FUNCTION_BLOCK FB_SoftWash IMPLEMENTS I_WashStrategy
VAR
	 stSettings : ST_WashSettings; 
    bStarted : BOOL := FALSE; 
END_VAR

METHOD FB_init : BOOL
VAR_INPUT
	bInitRetains : BOOL; // if TRUE, the retain variables are initialized (warm start / cold start)
	bInCopyCode : BOOL;  // if TRUE, the instance afterwards gets moved into the copy code (online change)
END_VAR
IF stSettings.sDescription = '' THEN 
    stSettings.rTemperature  := GVL_WashConstants.SOFT_TEMP; 
    stSettings.nSpinSpeed    := GVL_WashConstants.SOFT_SPIN; 
    stSettings.tWashDuration := GVL_WashConstants.SOFT_WASH_TIME; 
    stSettings.sDescription  := GVL_WashConstants.SOFT_DESC; 

END_IF 

 FB_init := TRUE;
END_METHOD

{warning 'add method implementation '}
METHOD GetDuration : TIME
  GetDuration := stSettings.tWashDuration;
END_METHOD

{warning 'add method implementation '}
METHOD GetProgramName : STRING
 GetProgramName := 'SOFT';
END_METHOD

{warning 'add method implementation '}
METHOD GetSettings : ST_WashSettings
  GetSettings := stSettings;
END_METHOD

{warning 'add method implementation '}
METHOD Start : BOOL
bStarted := TRUE; 
Start     := TRUE;
END_METHOD

END_FUNCTION_BLOCK

(* stored: Version 1.1.0.1, ProductVersion 3.1.4024.16
   POU FB_SoftWash: Id {20098e3f-b3d7-4b4d-bf5b-8d6ee14faa53}, SpecialFunc None
   Method FB_init: Id {a4b3b9de-443f-4248-aed5-d62c01d2d711}
   Method GetDuration: Id {87afdd7e-b00b-4cfb-a9ab-b46c0c02e1ff}
   Method GetProgramName: Id {55729a0a-7107-4950-a342-812a8f56501f}
   Method GetSettings: Id {81cfdbe6-36fa-42dd-a16c-4f0e926ac1f8}
   Method Start: Id {4f4c084b-101d-436b-b77f-113336563e31} *)
